// SIMATIC S7-200 project (STEP 7-Micro/WIN), CPU 222 REL 01.10

SYMBOL_TABLE SYM1
Terminal_Block_Error M0.0
Blown_Fuse_Error M0.1
No_User_Power_Error M0.2     // 无使用电源错误，该位置1
Out_of_Range_Error M0.3     // 模块范围溢出，该位置1
Parity_Error     M0.4
ID_0_Error       M0.5     // 扩展槽中没有EM231热电偶模块，该位置1
Module_0_Good    M0.6     // 无模块错误，该位置1
Configuration_Error M0.7     // 模块中有组态错误，该位置1
TC0_Image        VW0      // 该字中包括模拟量输入通道TC0的输入镜像
TC1_Image        VW2      // 该字中包括模拟量输入通道TC1的输入镜像
TC2_Image        VW4      // 该字中包括模拟量输入通道TC2的输入镜像
TC3_Image        VW6      // 该字中包括模拟量输入通道TC3的输入镜像
TC0              AIW0     // 该字中包括从热电偶0中读取的模拟量值
TC1              AIW2     // 该字中包括从热电偶1中读取的模拟量值
TC2              AIW4     // 该字中包括从热电偶2中读取的模拟量值
TC3              AIW6     // 该字中包括从热电偶3中读取的模拟量值
Always_On        SM0.0
First_Scan_On    SM0.1
END_SYMBOL_TABLE

ORGANIZATION_BLOCK MAIN:OB1
TITLE=
BEGIN
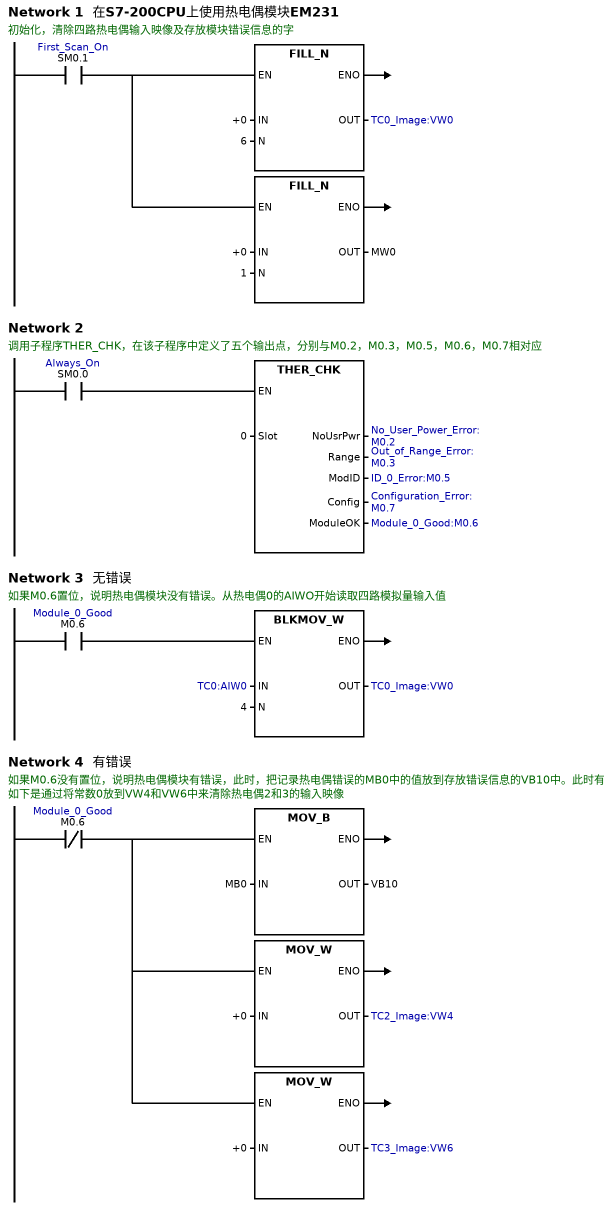
Network 1 // 在S7-200CPU上使用热电偶模块EM231
// 初始化，清除四路热电偶输入映像及存放模块错误信息的字
// Load SM0.1.
// Clear VW0 to VW10.
// Clear MW0.
LD     First_Scan_On:SM0.1
FILL   +0, TC0_Image:VW0, 6
FILL   +0, MW0, 1
Network 2
// 调用子程序THER_CHK，在该子程序中定义了五个输出点，分别与M0.2，M0.3，M0.5，M0.6，M0.7相对应
// Load SM0.0
// Call subroutine SBR0.
LD     Always_On:SM0.0
CALL   THER_CHK:SBR0, 0, No_User_Power_Error:M0.2, Out_of_Range_Error:M0.3, ID_0_Error:M0.5, Configuration_Error:M0.7, Module_0_Good:M0.6
Network 3 // 无错误
// 如果M0.6置位，说明热电偶模块没有错误。从热电偶0的AIWO开始读取四路模拟量输入值
//Load M0.6.
//Move good values to new location.
LD     Module_0_Good:M0.6
BMW    TC0:AIW0, TC0_Image:VW0, 4
Network 4 // 有错误
// 如果M0.6没有置位，说明热电偶模块有错误，此时，把记录热电偶错误的MB0中的值放到存放错误信息的VB10中。此时有两种选择：一是什么都不做来冻结热电偶信息，二是传送一个常数到热电偶信息中
// 如下是通过将常数0放到VW4和VW6中来清除热电偶2和3的输入映像
//Load M0.6 as a Normally Closed contact.
//Latch error information.
//Freeze Thermocouple0
//Freeze Thermocouple1
//Clear Thermocouple2.
//Clear Thermocouple3.
//NETWORK TITLE (single line)
//NETWORK COMMENTS
LDN    Module_0_Good:M0.6
MOVB   MB0, VB10
MOVW   +0, TC2_Image:VW4
MOVW   +0, TC3_Image:VW6
END_ORGANIZATION_BLOCK

SUBROUTINE_BLOCK THER_CHK:SBR0
TITLE=***SUBROUTINE***  THER_CHK
// 处理错误信息
VAR_INPUT
Slot:BYTE;	// LB0 
END_VAR
VAR_OUTPUT
NoUsrPwr:BOOL;	// L1.0 
Range:BOOL;	// L1.1 
ModID:BOOL;	// L1.2 
Config:BOOL;	// L1.3 
ModuleOK:BOOL;	// L1.4 
END_VAR
VAR
IDandErr:WORD;	// LW2 
END_VAR
BEGIN
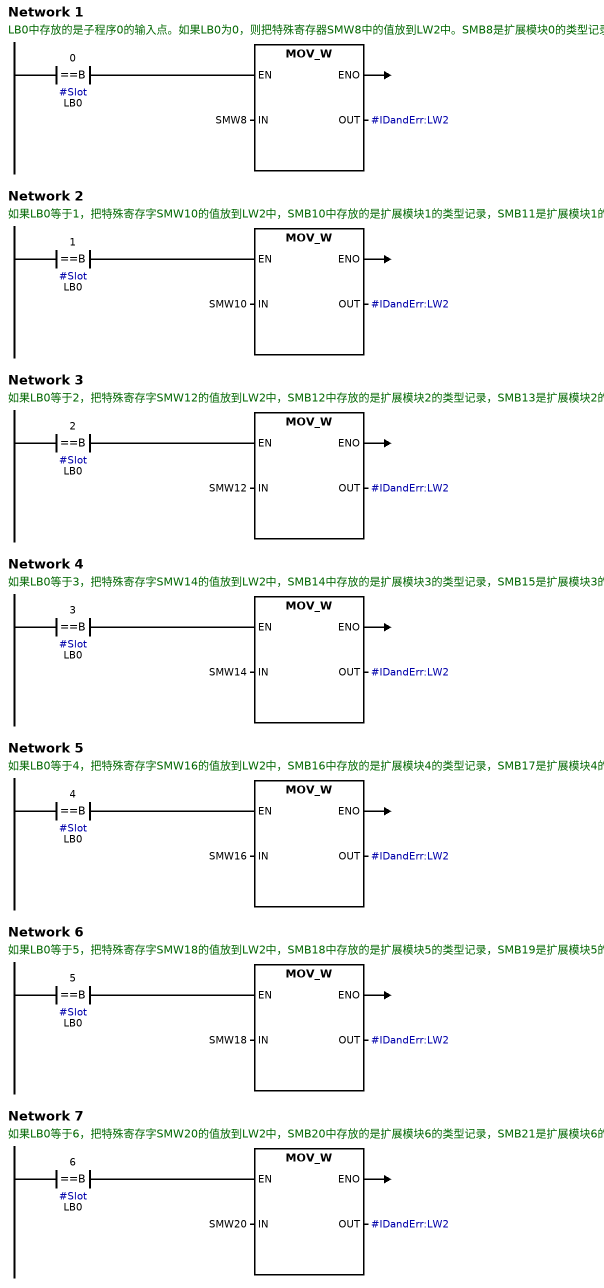
Network 1
// LB0中存放的是子程序0的输入点。如果LB0为0，则把特殊寄存器SMW8中的值放到LW2中。SMB8是扩展模块0的类型记录，SMB9是扩展模块0的错误记录
//Compare slot number to 0.
//Copy ID and Error info to LW2.
LDB=   0, #Slot:LB0
MOVW   SMW8, #IDandErr:LW2
Network 2
// 如果LB0等于1，把特殊寄存字SMW10的值放到LW2中，SMB10中存放的是扩展模块1的类型记录，SMB11是扩展模块1的错误记录
//Compare slot number to 1.
//Copy ID and Error info to LW2.
LDB=   1, #Slot:LB0
MOVW   SMW10, #IDandErr:LW2
Network 3
// 如果LB0等于2，把特殊寄存字SMW12的值放到LW2中，SMB12中存放的是扩展模块2的类型记录，SMB13是扩展模块2的错误记录
//Compare slot number to 2.
//Copy ID and Error info to LW2.
LDB=   2, #Slot:LB0
MOVW   SMW12, #IDandErr:LW2
Network 4
// 如果LB0等于3，把特殊寄存字SMW14的值放到LW2中，SMB14中存放的是扩展模块3的类型记录，SMB15是扩展模块3的错误记录
//Compare slot number to 3.
//Copy ID and Error info to LW2.
LDB=   3, #Slot:LB0
MOVW   SMW14, #IDandErr:LW2
Network 5
// 如果LB0等于4，把特殊寄存字SMW16的值放到LW2中，SMB16中存放的是扩展模块4的类型记录，SMB17是扩展模块4的错误记录
//Compare slot number to 4.
//Copy ID and Error info to LW2.
LDB=   4, #Slot:LB0
MOVW   SMW16, #IDandErr:LW2
Network 6
// 如果LB0等于5，把特殊寄存字SMW18的值放到LW2中，SMB18中存放的是扩展模块5的类型记录，SMB19是扩展模块5的错误记录
//Compare slot number to 5.
//Copy ID and Error info to LW2.
LDB=   5, #Slot:LB0
MOVW   SMW18, #IDandErr:LW2
Network 7
// 如果LB0等于6，把特殊寄存字SMW20的值放到LW2中，SMB20中存放的是扩展模块6的类型记录，SMB21是扩展模块6的错误记录
//Compare slot number to 6.
//Copy ID and Error info to LW2.
//Check for Module Errors Supported by Thermocouple
LDB=   6, #Slot:LB0
MOVW   SMW20, #IDandErr:LW2
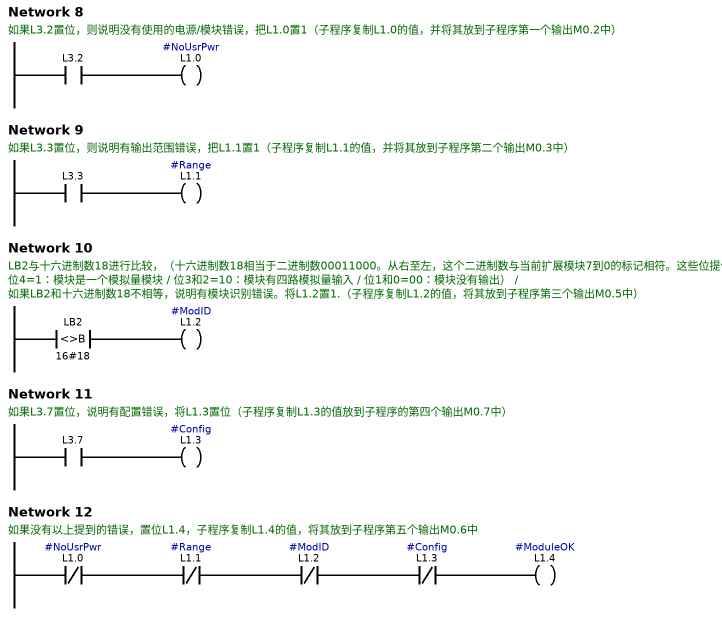
Network 8
//  如果L3.2置位，则说明没有使用的电源/模块错误，把L1.0置1（子程序复制L1.0的值，并将其放到子程序第一个输出M0.2中）
LD     L3.2
=      #NoUsrPwr:L1.0
Network 9
// 如果L3.3置位，则说明有输出范围错误，把L1.1置1（子程序复制L1.1的值，并将其放到子程序第二个输出M0.3中）
LD     L3.3
=      #Range:L1.1
Network 10
// LB2与十六进制数18进行比较，（十六进制数18相当于二进制数00011000。从右至左，这个二进制数与当前扩展模块7到0的标记相符。这些位提供了如下信息：
// 位7=0：说明有模块
// 位6和5=00：模块是非智能I/O模块
// 位4=1：模块是一个模拟量模块
// 位3和2=10：模块有四路模拟量输入
// 位1和0=00：模块没有输出）
// 如果LB2和十六进制数18不相等，说明有模块识别错误。将L1.2置1.（子程序复制L1.2的值，将其放到子程序第三个输出M0.5中）
LDB<>  LB2, 16#18
=      #ModID:L1.2
Network 11
// 如果L3.7置位，说明有配置错误，将L1.3置位（子程序复制L1.3的值放到子程序的第四个输出M0.7中）
LD     L3.7
=      #Config:L1.3
Network 12
// 如果没有以上提到的错误，置位L1.4，子程序复制L1.4的值，将其放到子程序第五个输出M0.6中
LDN    #NoUsrPwr:L1.0
AN     #Range:L1.1
AN     #ModID:L1.2
AN     #Config:L1.3
=      #ModuleOK:L1.4
END_SUBROUTINE_BLOCK
